Fanuc KAREL source: DISCTRL_FORM.kl

PROGRAM T
%NOLOCKGROUP
VAR
 v0 : STRING[40]
 v1 : INTEGER
 v2 : ARRAY[10] OF STRING[40]
 v3 : ARRAY[10] OF BOOLEAN
 v4 : ARRAY[10] OF BOOLEAN
 v5 : INTEGER
 v6 : INTEGER
 v7 : INTEGER
 v8 : INTEGER
BEGIN
 DISCTRL_FORM(v0, v1, v2, v3, v4, v5, v6, v7, v8)
END T
